_CFC_ (* Continuous Function Chart, elements in execution order *)
#0 RT_Pusk:R_TRIG(CLK: SHU6_P2_UST_RE_PUSK)
#1 TON_PCH_OTKL:TON(IN: SHU6_P2_UST_RE_STOP, PT: T#1s)
#2 FT_PCH_OTKL:R_TRIG(CLK: #1.Q)
#3 RS_YA2_Open:RS(SET: #0.Q, RESET1: #2.Q)
#4 ZADERJ_SHOD_YA2:TON(IN: #3.Q1, PT: t#10s)
#5 TON_YA2_Z_ZAM_TE4:TON(IN: SHU6_P2_TE4_M_ZASCH, PT: t#5s)
#6 AND(NOT SHU6_P2_SA1_DI1_A, NOT SHU6_P2_SA1_DI2_M)
#7 OR(SHU6_P2_Z_AV, #6)
#8 TON_OTK_MV:TON(IN: #7, PT: t#5s)
#9 OR(#5.Q, Z_ZAM_SR, #8.Q)
#10 SEL(SHU6_P2_YA2_SA6_DI7_A, eHVAC2PointActuatorMode_Close_OP, eHVAC2PointActuatorMode_Auto_BMS)
#11 SEL(#9, #10, eHVAC2PointActuatorMode_Close_OP)
#12 fb_HVACPA:FB_HVAC2PointActuator(eHVACDataSecurityType_Idle, FALSE, TRUE, #4.Q, #11, SHU6_P2_KV1_DI8, SHU6_P2_YA2_DI3_ZKR, SHU6_P2_YA2_DI4_OTK, TRUE, SHU6_P2_SB, enableLimitSwitch, stokeTime)
#13 SHU6_P2_YA2_DO2_OTK <= #12.out 1
#14 OR(#12.out 4, #12.out 5)
#15 YA2_OTKAZ <= #14
#16 INT_TO_TIME(SHU6_P2_YA2_VREMYA_HODA)
#17 MUL(#16, 1000)
#18 stokeTime <= #17
_END_CFC_
END_PROGRAM

(* POU IM/YA3_Upr, CFC *)
PROGRAM YA3_Upr
VAR
	YA3_PID: FB_HVACPIDCtrl;

	deadRange: REAL := 0.1;
	direction: BOOL;
	tTi: TIME;
	tTv: TIME;
	tTd: TIME;

	rYMin: REAL := 0;
	rYMax: REAL := 100;
	TON_SHU6_P2_P1_DI7_RUN: TON;
	reg1: BOOL;
	reg2: BOOL;

	SHU6_P2_YA3_: BOOL;
	YA3_REG_POL: BOOL;
	rwx: REAL;
	EPS1: REAL;
	EPS2: REAL;
END_VAR
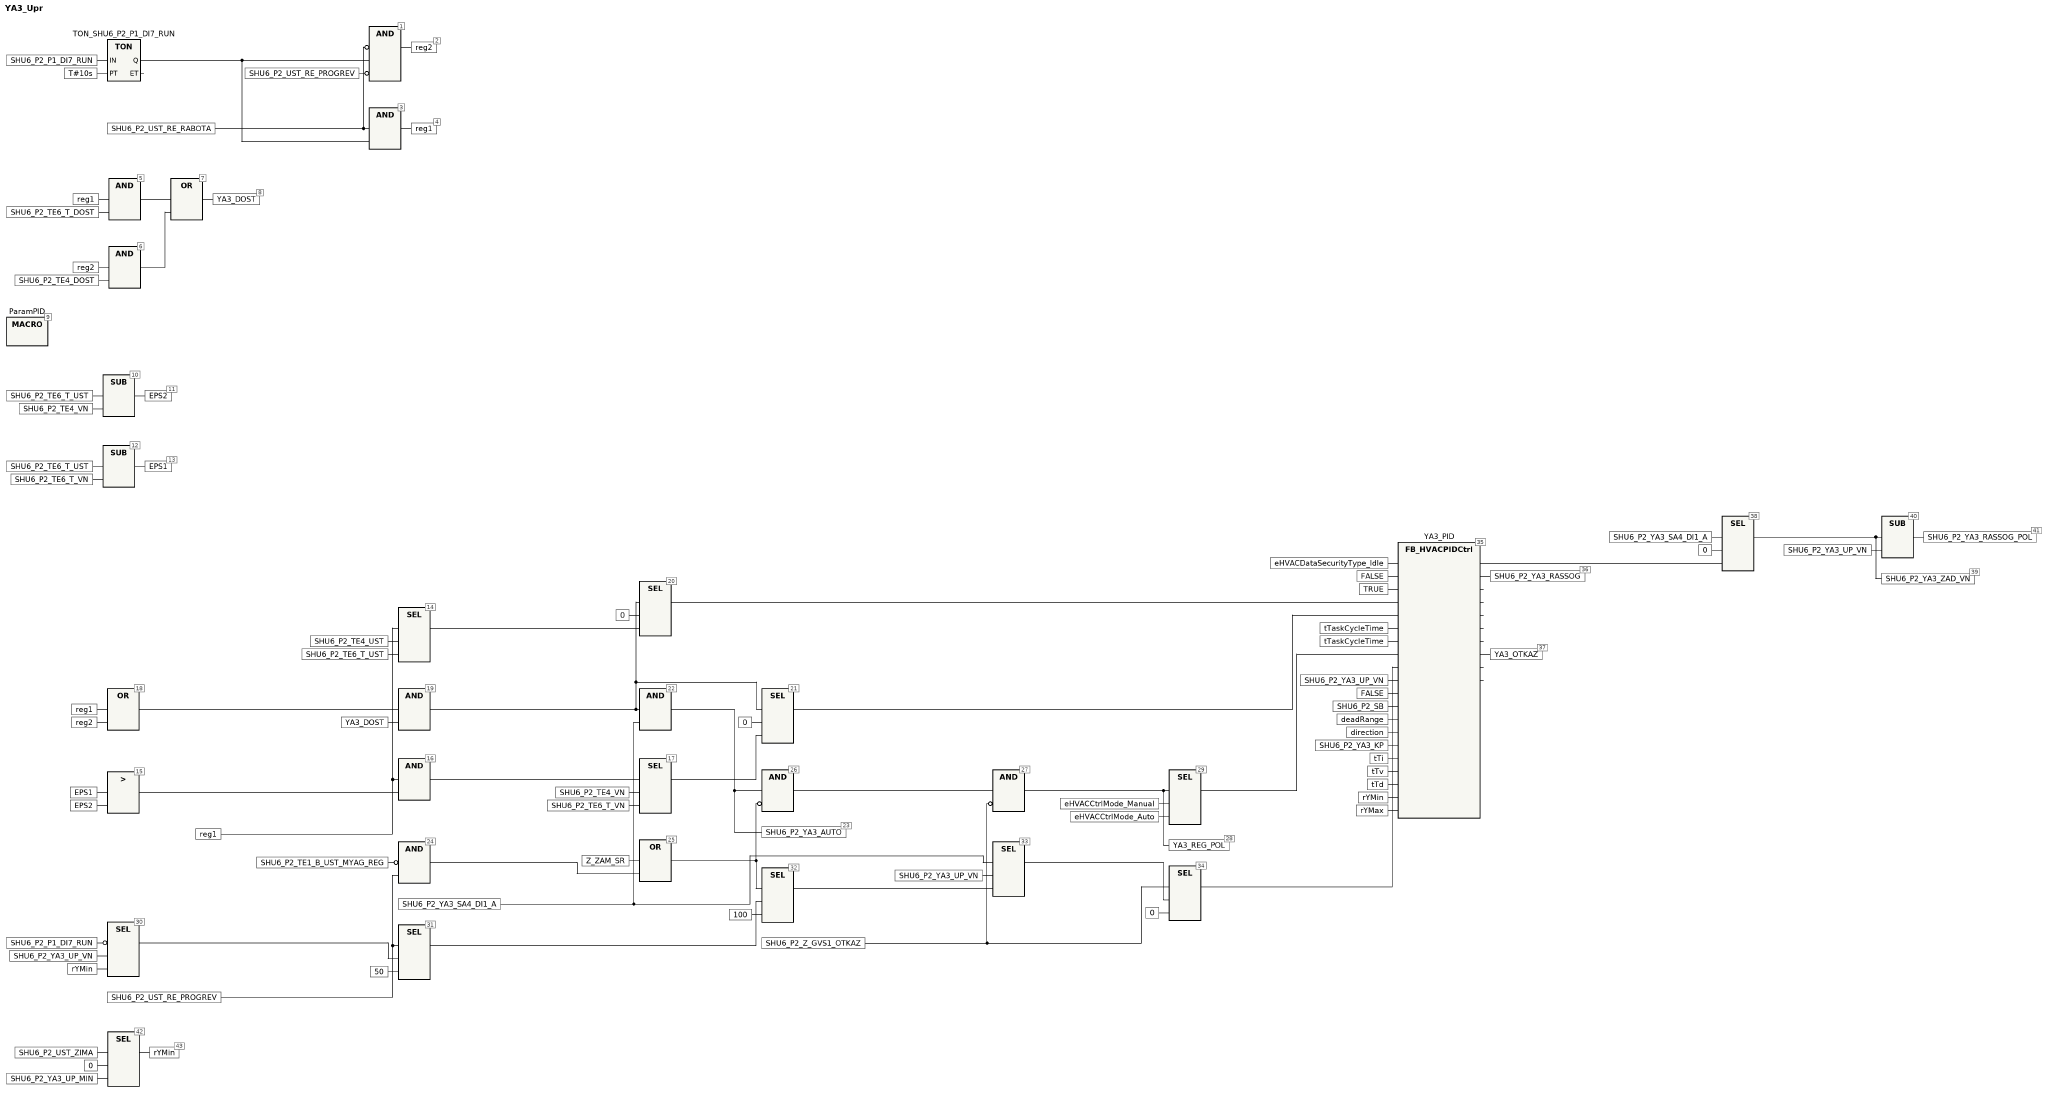
